Fanuc KAREL source: ko00008.KL

-- PROVISIONAL review KL for V1013-1; original PC SHA256 3314dc1bce4e1df0dbc5358165c95bf3cb3b03b985aa85c0d560ad3b3a0e080b
-- Incomplete behavior may be omitted. Consult companion uncertainty JSON. Do not deploy.
PROGRAM KO00008
%NOLOCKGROUP
-- UNRESOLVED_DECL P1 type=000101
-- UNRESOLVED_DECL P2 type=000101
-- UNRESOLVED_DECL P3 type=000101
-- UNRESOLVED_DECL P4 type=000101
-- UNRESOLVED_DECL OUT type=000199
BEGIN
  -- UNRESOLVED_PC offsets 5-68; opcodes 27,22,1C,22,1C,22,1C,22,1C,76,7E,4A
  -- UNRESOLVED_PC offsets 73-77; opcodes 7F
END KO00008
